// TIA Portal V19 export
FUNCTION_BLOCK "PitTable1_FB"   // FB166, LAD
TITLE = PIT TABLE LOOP PNEUMATIC
// stored: MemoryReserve 100, SetENOAutomatically false
   VAR_INPUT
      AreaInterface : "AreaInterface";
      ZSI : "udt_ZoneSafetyInterface";
      DSI : "udt_DeviceSafetyInterface";
      DataIn : Struct
         Pb_Up : Bool;
         Pb_Dwn : Bool;
         Ls_Up : Bool;
         Ls_Down : Bool;
      END_STRUCT;
      CIn : Struct
         Manager : "ValveMachine_Manager";
         ExtEnable_Up : Bool;
         ExtEnable_Down : Bool;
      END_STRUCT;
      Config : Struct
         LIFT : "ValveMachine_Config";
         Exist : Bool;
      END_STRUCT;
   END_VAR
   VAR_OUTPUT
      MachineInterface : "MachineInterface";
      DataOut : Struct
         V_Up : Bool;
         V_Down : Bool;
         Lamp : Bool;
      END_STRUCT;
   END_VAR
   VAR
      Warning : "ValveMachine_Wng";
      Alarm : "ValveAlr";
      Lift : "ValveMachine_FB";
      TimerRestManualReq : TON_TIME;
   END_VAR
   VAR_TEMP
      Dummy : Bool;
   END_VAR
BEGIN

REGION Network 1: DataIn
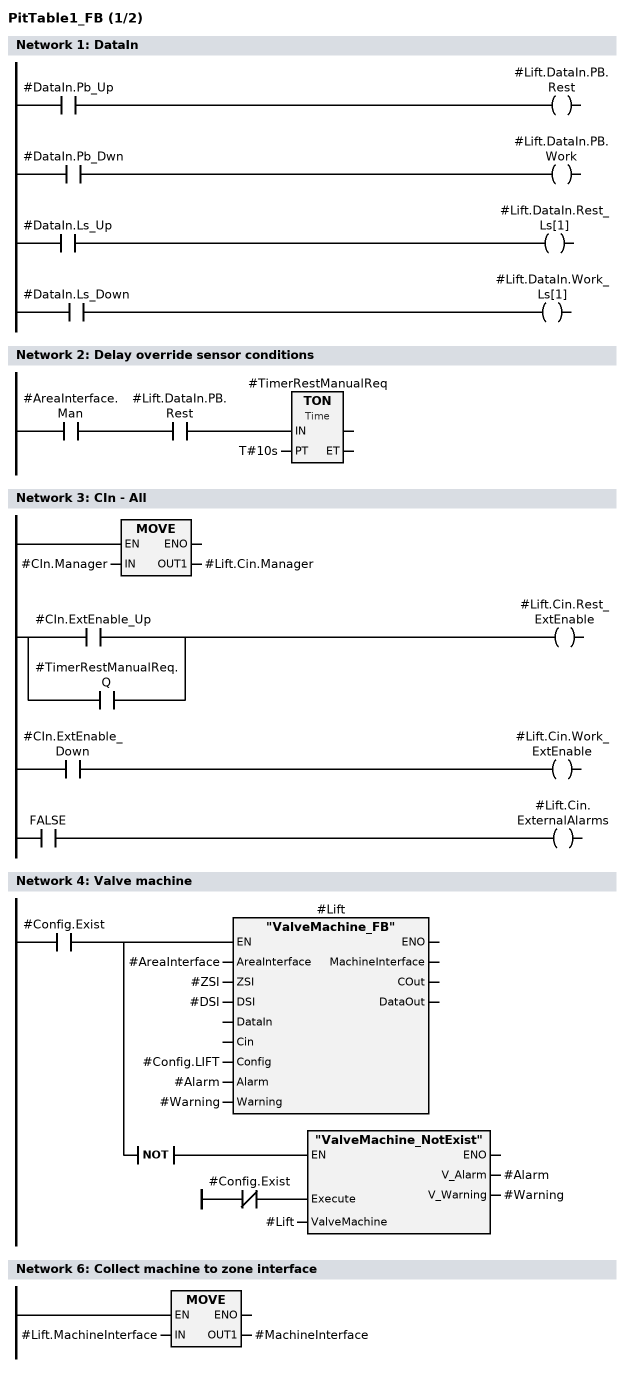
   RUNG wire#powerrail
      Contact( #DataIn.Pb_Up )
      Coil( #Lift.DataIn.PB.Rest )
   END_RUNG
   RUNG wire#powerrail
      Contact( #DataIn.Pb_Dwn )
      Coil( #Lift.DataIn.PB.Work )
   END_RUNG
   RUNG wire#powerrail
      Contact( #DataIn.Ls_Up )
      Coil( #Lift.DataIn.Rest_Ls[1] )
   END_RUNG
   RUNG wire#powerrail
      Contact( #DataIn.Ls_Down )
      Coil( #Lift.DataIn.Work_Ls[1] )
   END_RUNG
   // the same network as SCL:
   #Lift.DataIn.PB.Rest := #DataIn.Pb_Up;
   #Lift.DataIn.PB.Work := #DataIn.Pb_Dwn;
   #Lift.DataIn.Rest_Ls[1] := #DataIn.Ls_Up;
   #Lift.DataIn.Work_Ls[1] := #DataIn.Ls_Down;
END_REGION

REGION Network 2: Delay override sensor conditions
   RUNG wire#powerrail
      Contact( #AreaInterface.Man )
      Contact( #Lift.DataIn.PB.Rest )
      { S7_Templates := "time_type := Time" } #TimerRestManualReq.TON(pt := T#10s, et =>)
   END_RUNG
   // the same network as SCL:
   #TimerRestManualReq(IN := #AreaInterface.Man AND #Lift.DataIn.PB.Rest, PT := T#10s);   // TON
END_REGION

REGION Network 3: CIn - All
   RUNG wire#powerrail
      Move(in := #CIn.Manager, out1 => #Lift.Cin.Manager)
   END_RUNG
   RUNG wire#powerrail
      Contact( #CIn.ExtEnable_Up )
      wire#w1
      Coil( #Lift.Cin.Rest_ExtEnable )
   END_RUNG
   RUNG wire#powerrail
      Contact( #TimerRestManualReq.Q )
   END_RUNG wire#w1
   RUNG wire#powerrail
      Contact( #CIn.ExtEnable_Down )
      Coil( #Lift.Cin.Work_ExtEnable )
   END_RUNG
   RUNG wire#powerrail
      Contact( FALSE )
      Coil( #Lift.Cin.ExternalAlarms )
   END_RUNG
   // the same network as SCL:
   #Lift.Cin.Manager := #CIn.Manager;
   #Lift.Cin.Rest_ExtEnable := #CIn.ExtEnable_Up OR #TimerRestManualReq.Q;
   #Lift.Cin.Work_ExtEnable := #CIn.ExtEnable_Down;
   #Lift.Cin.ExternalAlarms := FALSE;
END_REGION

REGION Network 4: Valve machine
   RUNG wire#powerrail
      Contact( #Config.Exist )
      wire#w1
      #Lift(AreaInterface := #AreaInterface, ZSI := #ZSI, DSI := #DSI, DataIn :=, Cin :=, Config := #Config.LIFT, Alarm := #Alarm, Warning := #Warning, MachineInterface =>, COut =>, DataOut =>)
   END_RUNG
   RUNG wire#w1
      Not()
      "ValveMachine_NotExist"(Execute := wire#w2, ValveMachine := #Lift, V_Alarm => #Alarm, V_Warning => #Warning)
   END_RUNG
   RUNG wire#powerrail
      I_Contact( #Config.Exist )
   END_RUNG wire#w2
   // the same network as SCL:
   IF #Config.Exist THEN
       #Lift(AreaInterface := #AreaInterface,   // "ValveMachine_FB"
             ZSI := #ZSI,
             DSI := #DSI,
             Config := #Config.LIFT,
             Alarm := #Alarm,
             Warning := #Warning);
   END_IF;
   IF NOT #Config.Exist THEN
       "ValveMachine_NotExist"(Execute := NOT #Config.Exist,
                               ValveMachine := #Lift,
                               V_Alarm => #Alarm,
                               V_Warning => #Warning);
   END_IF;
END_REGION

REGION Network 5: <<< MACHINE STATUS >>>
END_REGION

REGION Network 6: Collect machine to zone interface
   RUNG wire#powerrail
      Move(in := #Lift.MachineInterface, out1 => #MachineInterface)
   END_RUNG
   // the same network as SCL:
   #MachineInterface := #Lift.MachineInterface;
END_REGION

REGION Network 7: Data out (Valve solenoid)
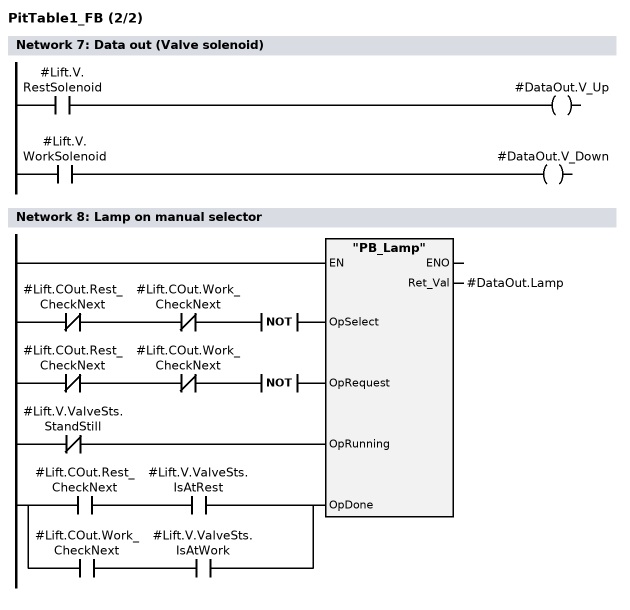
   RUNG wire#powerrail
      Contact( #Lift.V.RestSolenoid )
      Coil( #DataOut.V_Up )
   END_RUNG
   RUNG wire#powerrail
      Contact( #Lift.V.WorkSolenoid )
      Coil( #DataOut.V_Down )
   END_RUNG
   // the same network as SCL:
   #DataOut.V_Up := #Lift.V.RestSolenoid;
   #DataOut.V_Down := #Lift.V.WorkSolenoid;
END_REGION

REGION Network 8: Lamp on manual selector
   RUNG wire#powerrail
      "PB_Lamp"(OpSelect := wire#w1, OpRequest := wire#w2, OpRunning := wire#w3, OpDone := wire#w4, Ret_Val => #DataOut.Lamp)
   END_RUNG
   RUNG wire#powerrail
      I_Contact( #Lift.COut.Rest_CheckNext )
      I_Contact( #Lift.COut.Work_CheckNext )
      Not()
   END_RUNG wire#w1
   RUNG wire#powerrail
      I_Contact( #Lift.COut.Rest_CheckNext )
      I_Contact( #Lift.COut.Work_CheckNext )
      Not()
   END_RUNG wire#w2
   RUNG wire#powerrail
      I_Contact( #Lift.V.ValveSts.StandStill )
   END_RUNG wire#w3
   RUNG wire#powerrail
      Contact( #Lift.COut.Rest_CheckNext )
      Contact( #Lift.V.ValveSts.IsAtRest )
   END_RUNG wire#w4
   RUNG wire#powerrail
      Contact( #Lift.COut.Work_CheckNext )
      Contact( #Lift.V.ValveSts.IsAtWork )
   END_RUNG wire#w4
   // the same network as SCL:
   #DataOut.Lamp := "PB_Lamp"(OpSelect := NOT (NOT #Lift.COut.Rest_CheckNext AND NOT #Lift.COut.Work_CheckNext),
                           OpRequest := NOT (NOT #Lift.COut.Rest_CheckNext AND NOT #Lift.COut.Work_CheckNext),
                           OpRunning := NOT #Lift.V.ValveSts.StandStill,
                           OpDone := (#Lift.COut.Rest_CheckNext AND #Lift.V.ValveSts.IsAtRest) OR (#Lift.COut.Work_CheckNext AND #Lift.V.ValveSts.IsAtWork));
END_REGION
END_FUNCTION_BLOCK
